Fanuc KAREL source: kt00080.KL

-- PROVISIONAL review KL for V1013-1; original PC SHA256 879ccd2be373b097213e4b8712864bde8b28daa725b14bd93bb56ac9823f8815
-- Incomplete behavior may be omitted. Consult companion uncertainty JSON. Do not deploy.
PROGRAM KT00080
%NOLOCKGROUP
VAR
  R1 : REAL
  OUT : REAL
-- UNRESOLVED_DECL H2 type=002017
BEGIN
  -- UNRESOLVED_PC offsets 5-16; opcodes 2E,23
  -- UNRESOLVED_PC offsets 21-35; opcodes 2E,22,9D,33,B4
  -- UNRESOLVED_PC offsets 40-63; opcodes 21,22,9D,33,B3,64,6B,23
  -- UNRESOLVED_PC offsets 68-72; opcodes 7F
END KT00080
